{attribute 'qualified_only'}
VAR_GLOBAL CONSTANT
    MAX_SHUTTER_OUTPUTS : INT := 1;
	MAX_LIGHT_OUTPUTS_PER_LEVEL : INT := 3;
	MAX_SIMPLE_OUTPUTS : INT := 3;
	MAX_SHUTTERS : INT := 11;
	MAX_LIGHTS : INT := 1;//TODO 50 ALBO MNIEJ;
	MAX_SIMPLE_BUTTONS : INT := 3; //TODO PEWNIE WIECEJ
END_VAR

VAR_GLOBAL
	
	din_1_1_1 AT %I* : BOOL; //garaż po prawej stronie od drzwi
	din_1_2_2 AT %I* : BOOL; //garaż po lewej stronie od drzwi (wh-gn->bl) + pralnia po lewej stronie od drzwi, pierwszy od dołu (trzeba namierzyć)
	din_1_3_3 AT %I* : BOOL; //pralnia po lewej stronie od drzwi, drugi od dołu (trzeba namierzyć)
	din_1_4_4 AT %I* : BOOL; 
	din_1_5_5 AT %I* : BOOL;
	din_1_6_6 AT %I* : BOOL; 
	din_1_7_7 AT %I* : BOOL;
	din_1_8_8 AT %I* : BOOL;
	din_1_9_9 AT %I* : BOOL; 
	din_05zModulu1_przewod_5_s_27_1_pralnia_1z2_pomaranczowy AT %I* : BOOL; //zasilanie bialo-zielony: Wlacznik roletowy w pralni gora
	din_04zModulu1_przewod_5_s_27_1_pralnia_2z2_niebieski AT %I* : BOOL; //zasilanie bialo-zielony: Wlacznik roletowy w pralni dol

	din_04zModulu2_przewod_3_s_30_1_kuchnia_1z2_niebieski  AT %I* : BOOL; //zasilanie bialo-zielony: Wlacznik roletowy w kuchni kuchnia dol
	din_03zModulu2_przewod_3_s_30_1_kuchnia_2z2_zielony  AT %I* : BOOL; //zasilanie bialo-zielony: Wlacznik roletowy w kuchni kuchnia gora
    
    din_06zModulu2_przewod_3_s_30_1_kuchnia_1z2_brazowy  AT %I* : BOOL; //zasilanie bialo-zielony: Wlacznik roletowy w kuchni wykusz gora
	din_05zModulu2_przewod_3_s_30_1_kuchnia_2z2_pomaranczowy  AT %I* : BOOL; //zasilanie bialo-zielony: Wlacznik roletowy w kuchni wykusz dol

    din_08zModulu2_przewod_3_s_30_1_kuchnia_1z2_bialopomaranczowy  AT %I* : BOOL; //zasilanie bialo-zielony: Wlacznik roletowy w kuchni slide gora
	din_07zModulu2_przewod_3_s_30_1_kuchnia_2z2_bialoniebieski  AT %I* : BOOL; //zasilanie bialo-zielony: Wlacznik roletowy w kuchni slide dol

    din_03zModulu3_przewod_14_s_26_1_gabinet_1z2_pomaranczowy  AT %I* : BOOL; //zasilanie bialo-zielony: Wlacznik roletowy w gabinecie gora
	din_02zModulu3_przewod_14_s_26_1_gabinet_2z2_niebieski  AT %I* : BOOL; //zasilanie bialo-zielony: Wlacznik roletowy w gabinecie dol
	

	din_10zModulu1_przewod_1_s_25_1_koniecPrzedpokojuElektronicznyPoczworny_1z4_brazowy AT %I* : BOOL;//bylo din1_10_10 //zasilanie biało-zielony: Elektroniczny wlacznik swiatla w przedpokoju 1/4 lub wlacznik poczworny w kuchni na slupku
	din_11zModulu1_przewod_1_s_25_1_koniecPrzedpokojuElektronicznyPoczworny_2z4_bialoniebieski AT %I* : BOOL; //bylo din1_11_11 //zasilanie biało-zielony: Elektroniczny wlacznik swiatla w przedpokoju 2/4
	din_12zModulu1_przewod_1_s_25_1_koniecPrzedpokojuElektronicznyPoczworny_3z4_bialopomaranczowy AT %I* : BOOL; //bylo din1_12_12 //zasilanie biało-zielony: Elektroniczny wlacznik swiatla w przedpokoju 3/4 lub wlacznik poczworny na dole schodow 1/4
	din_13zModulu1_przewod_xxxxxxxx_koniecPrzedpokojuElektronicznyPoczworny_4z4_bialobrazowy AT %I* : BOOL; //din_1_13_13 //zasilanie bialo-zielony: Elektroniczny wlacznik swiatla w przedpokoju 4/4	

	
	din_1_14_14 AT %I* : BOOL;
	din_1_15_15 AT %I* : BOOL;
	din_1_16_16 AT %I* : BOOL;

	CsvPersistentEventStorage : FB_CsvPersistentEventStorage;
	EventLogger : EventLogger(CsvPersistentEventStorage);
	

//-------------------------------------------------------------------------------------------------	
//OUTPUTS
	dout_1_zaluzja_pralnia_w_gore AT %Q* : BOOL;
	douts_1_zaluzja_pralnia_w_gore : ARRAY[1..MAX_SHUTTER_OUTPUTS] OF BOOL; 	
	dout_2_zaluzja_pralnia_w_dol AT %Q* : BOOL;
	douts_2_zaluzja_pralnia_w_dol : ARRAY[1..MAX_SHUTTER_OUTPUTS] OF BOOL;
	
	dout_3_zaluzja_okno_narozne_kuchnia_w_gore AT %Q* : BOOL;
	douts_3_zaluzja_okno_narozne_kuchnia_w_gore : ARRAY[1..MAX_SHUTTER_OUTPUTS] OF BOOL;
	dout_4_zaluzja_okno_narozne_kuchnia_w_dol AT %Q* : BOOL;
	douts_4_zaluzja_okno_narozne_kuchnia_w_dol : ARRAY[1..MAX_SHUTTER_OUTPUTS] OF BOOL;
	
	dout_5_zaluzja_wykusz_w_gore AT %Q* : BOOL;	
	douts_5_zaluzja_wykusz_w_gore : ARRAY[1..MAX_SHUTTER_OUTPUTS] OF BOOL; 
	dout_6_zaluzja_wykusz_w_dol AT %Q* : BOOL;
	douts_6_zaluzja_wykusz_w_dol : ARRAY[1..MAX_SHUTTER_OUTPUTS] OF BOOL;
	
	dout_7_zaluzja_slide_w_gore AT %Q* : BOOL;	
	douts_7_zaluzja_slide_w_gore : ARRAY[1..MAX_SHUTTER_OUTPUTS] OF BOOL; 
	dout_8_zaluzja_slide_w_dol AT %Q* : BOOL;
	douts_8_zaluzja_slide_w_dol : ARRAY[1..MAX_SHUTTER_OUTPUTS] OF BOOL;
	
	dout_9_zaluzja_gabinet_w_gore AT %Q* : BOOL;	
	douts_9_zaluzja_gabinet_w_gore : ARRAY[1..MAX_SHUTTER_OUTPUTS] OF BOOL; 
	dout_10_zaluzja_gabinet_w_dol AT %Q* : BOOL;
	douts_10_zaluzja_gabinet_w_dol : ARRAY[1..MAX_SHUTTER_OUTPUTS] OF BOOL;
	
	dout_11_zaluzja_balkon_w_gore AT %Q* : BOOL;	
	douts_11_zaluzja_balkon_w_gore : ARRAY[1..MAX_SHUTTER_OUTPUTS] OF BOOL; 
	dout_12_zaluzja_balkon_w_dol AT %Q* : BOOL;	
	douts_12_zaluzja_balkon_w_dol : ARRAY[1..MAX_SHUTTER_OUTPUTS] OF BOOL; 
	
	dout_13_zaluzja_nad_wykuszem_w_gore AT %Q* : BOOL;
	douts_13_zaluzja_nad_wykuszem_w_gore : ARRAY[1..MAX_SHUTTER_OUTPUTS] OF BOOL;
	dout_14_zaluzja_nad_wykuszem_w_dol AT %Q* : BOOL;
	douts_14_zaluzja_nad_wykuszem_w_dol : ARRAY[1..MAX_SHUTTER_OUTPUTS] OF BOOL;
	
	dout_15_zaluzja_okno_bez_balkonu_w_gore AT %Q* : BOOL;	
	douts_15_zaluzja_okno_bez_balkonu_w_gore : ARRAY[1..MAX_SHUTTER_OUTPUTS] OF BOOL; 
	dout_16_zaluzja_okno_bez_balkonu_w_dol AT %Q* : BOOL;
	douts_16_zaluzja_okno_bez_balkonu_w_dol : ARRAY[1..MAX_SHUTTER_OUTPUTS] OF BOOL;
	
	dout_17_roleta_kotlownia_w_gore AT %Q* : BOOL;	
	douts_17_roleta_kotlownia_w_gore : ARRAY[1..MAX_SHUTTER_OUTPUTS] OF BOOL; 
	dout_18_roleta_kotlownia_w_dol AT %Q* : BOOL;
	douts_18_roleta_kotlownia_w_dol : ARRAY[1..MAX_SHUTTER_OUTPUTS] OF BOOL;
	
	dout_19_roleta_warsztat_w_gore AT %Q* : BOOL;	
	douts_19_roleta_warsztat_w_gore : ARRAY[1..MAX_SHUTTER_OUTPUTS] OF BOOL; 
	dout_20_roleta_warsztat_w_dol AT %Q* : BOOL;
	douts_20_roleta_warsztat_w_dol : ARRAY[1..MAX_SHUTTER_OUTPUTS] OF BOOL;
	
	dout_21_roleta_kotlownia_w_gore AT %Q* : BOOL;	
	douts_21_roleta_kotlownia_w_gore : ARRAY[1..MAX_SHUTTER_OUTPUTS] OF BOOL; 
	dout_22_roleta_kotlownia_w_dol AT %Q* : BOOL;
	douts_22_roleta_kotlownia_w_dol : ARRAY[1..MAX_SHUTTER_OUTPUTS] OF BOOL;
	
	

	dout_1zModulu1_przewod_2_o_4_1_swiatloSalonJadalniaSufit AT %Q* : BOOL; //2-o-4-1
		douts_swiatloSalonJadalniaSufit : ARRAY[1..MAX_LIGHT_OUTPUTS_PER_LEVEL] OF BOOL;
	dout_2zModulu1_przewod_2_o_5_1_swiatloSalonKanapaSufit AT %Q* : BOOL; //2-o-5-1
		douts_swiatloSalonKanapaSufit : ARRAY[1..MAX_LIGHT_OUTPUTS_PER_LEVEL] OF BOOL;
	dout_3zModulu1_przewod_2_o_7_1_swiatloPrzejscieZPrzedpokojuDoSalonuSufit AT %Q* : BOOL; //2-o-7-1
		douts_swiatloPrzejscieZPrzedpokojuDoSalonuSufit : ARRAY[1..MAX_LIGHT_OUTPUTS_PER_LEVEL] OF BOOL;
	dout_4zModulu1_przewod_x_o_x_x_swiatloSrodekSalonuSufit AT %Q* : BOOL; //xxxxx
		douts_swiatloSrodekSalonuSufit : ARRAY[1..MAX_LIGHT_OUTPUTS_PER_LEVEL] OF BOOL;
    
	dout_xxxxxxxx_przewod_xxxxxx_swiatloKontuarKuchnia AT %Q* : BOOL; //xxxxx
		douts_swiatloKontuarKuchnia : ARRAY[1..MAX_LIGHT_OUTPUTS_PER_LEVEL] OF BOOL;
	dout_xxxxxxxx_przewod_xxxxxx_swiatloKuchniaSufit AT %Q* : BOOL; //xxxxx
		douts_swiatloKuchniaSufit : ARRAY[1..MAX_LIGHT_OUTPUTS_PER_LEVEL] OF BOOL;
	dout_xxxxxxxx_przewod_xxxxxx_swiatloKuchniaPodSzafkami AT %Q* : BOOL; //xxxxx
		douts_swiatloKuchniaPodSzafkami : ARRAY[1..MAX_LIGHT_OUTPUTS_PER_LEVEL] OF BOOL;
	dout_xxxxxxxx_przewod_xxxxxx_swiatloPrzedpokojBlizejSalonu AT %Q* : BOOL; //xxxxx
		douts_swiatloPrzedpokojBlizejSalonu : ARRAY[1..MAX_LIGHT_OUTPUTS_PER_LEVEL] OF BOOL;
	dout_xxxxxxxx_przewod_xxxxxx_swiatloPrzedpokojBlizejDrzwi AT %Q* : BOOL; //xxxxx
		douts_swiatloPrzedpokojBlizejDrzwi : ARRAY[1..MAX_LIGHT_OUTPUTS_PER_LEVEL] OF BOOL;
	dout_xxxxxxxx_przewod_xxxxxx_swiatloTrepy AT %Q* : BOOL; //xxxxx
		douts_swiatloTrepy : ARRAY[1..MAX_LIGHT_OUTPUTS_PER_LEVEL] OF BOOL;
	dout_xxxxxxxx_przewod_xxxxxx_swiatloKorytarzPunktySufit AT %Q* : BOOL; //xxxxx
		douts_swiatloKorytarzPunktySufit : ARRAY[1..MAX_LIGHT_OUTPUTS_PER_LEVEL] OF BOOL;
	dout_xxxxxxxx_przewod_xxxxxx_swiatloZyrandolKorytarz AT %Q* : BOOL; //xxxxx
		douts_swiatloZyrandolKorytarz : ARRAY[1..MAX_LIGHT_OUTPUTS_PER_LEVEL] OF BOOL;
	dout_xxxxxxxx_przewod_xxxxxx_swiatloPralnia AT %Q* : BOOL; //xxxxx
		douts_swiatloPralnia : ARRAY[1..MAX_LIGHT_OUTPUTS_PER_LEVEL] OF BOOL;
	dout_xxxxxxxx_przewod_xxxxxx_swiatloToaletkaSypialniaRodzicow AT %Q* : BOOL; //xxxxx
		douts_swiatloToaletkaSypialniaRodzicow : ARRAY[1..MAX_LIGHT_OUTPUTS_PER_LEVEL] OF BOOL;
	dout_xxxxxxxx_przewod_xxxxxx_swiatlo AT %Q* : BOOL; //xxxxx
		douts_swiatloNiskiSufitSypialniaRodzicow : ARRAY[1..MAX_LIGHT_OUTPUTS_PER_LEVEL] OF BOOL;
	dout_xxxxxxxx_przewod_xxxxxx_swiatloNiskiSufitSypialniaRodzicow AT %Q* : BOOL; //xxxxx
		douts_swiatloWysokiSufitSypialniaRodzicow : ARRAY[1..MAX_LIGHT_OUTPUTS_PER_LEVEL] OF BOOL;
	dout_xxxxxxxx_przewod_xxxxxx_swiatloWysokiSufitSypialniaRodzicow AT %Q* : BOOL; //xxxxx
		douts_swiatlo : ARRAY[1..MAX_LIGHT_OUTPUTS_PER_LEVEL] OF BOOL;
	dout_xxxxxxxx_przewod_xxxxxx_swiatloNadLozkiemSypialniaRodzicow AT %Q* : BOOL; //xxxxx
		douts_swiatloNadLozkiemSypialniaRodzicow : ARRAY[1..MAX_LIGHT_OUTPUTS_PER_LEVEL] OF BOOL;
	dout_xxxxxxxx_przewod_xxxxxx_swiatloPrzedDomem AT %Q* : BOOL; //xxxxx
		douts_swiatloPrzedDomem : ARRAY[1..MAX_LIGHT_OUTPUTS_PER_LEVEL] OF BOOL;
	dout_xxxxxxxx_przewod_xxxxxx_swiatloPodbitki AT %Q* : BOOL; //xxxxx
		douts_swiatloPodbitki : ARRAY[1..MAX_LIGHT_OUTPUTS_PER_LEVEL] OF BOOL;
	dout_xxxxxxxx_przewod_xxxxxx_swiatloGaraz AT %Q* : BOOL; //xxxxx
		douts_swiatloGaraz : ARRAY[1..MAX_LIGHT_OUTPUTS_PER_LEVEL] OF BOOL;
	
	
END_VAR

(* stored: Version 1.1.0.1, ProductVersion 3.1.4024.12
   GVL GVL: Id {798ee332-7b17-4a9d-a450-87f1f742e8e3} *)
